// TIA Portal V17 export
// export: Created 2023-02-13T11:16:28.8867509Z, ExportSetting WithDefaults, DisplayName Totally Integrated Automation Portal, DisplayVersion V17, DisplayName TIA Portal Openness, DisplayVersion V17, DisplayName TIA Portal Teamcenter Gateway, DisplayVersion V17, DisplayName TIA Portal Version Control Interface, DisplayVersion V17, DisplayName SINAMICS Startdrive Advanced, DisplayVersion V17, DisplayName SINAMICS Startdrive G130, G150, S120, S150, SINAMICS MV, S210, DisplayVersion V17, DisplayName SINAMICS Startdrive G110M, G120, G120C, G120D, G120P, G115D, DisplayVersion V17, DisplayName STEP 7 Professional, DisplayVersion V17, DisplayName STEP 7 Safety, DisplayVersion V17, DisplayName WinCC Professional, DisplayVersion V17
FUNCTION_BLOCK "IO Digital Preparation"   // FB8, LAD
{ S7_Optimized_Access := 'FALSE' }
VERSION : 0.1
// stored: AutoNumber true, IsIECCheckEnabled false, SetENOAutomatically false, UDAEnableTagReadback false
   VAR_INPUT
      init : Bool;
      Reset : Bool;
   END_VAR
   VAR
      "FS-01.01" { S7_SetPoint := 'True'} : "Digital";   // FLOW SWITCH LINE HOT WATER PHE-01.01
      "DRP-P02.01" { S7_SetPoint := 'True'} : "Digital";   // DRY RUN PROTECTION MONO PUMP P-02.01
      "DRP-P02.02" { S7_SetPoint := 'True'} : "Digital";   // DRY RUN PROTECTION MONO PUMP P-02.03
      "DRP-P03.01" { S7_SetPoint := 'True'} : "Digital";   // DRY RUN PROTECTION MONO PUMP P-03.01
      "DRP-P03.02" { S7_SetPoint := 'True'} : "Digital";   // DRY RUN PROTECTION MONO PUMP P-03.03
      "DRP-P04.01" { S7_SetPoint := 'True'} : "Digital";   // DRY RUN PROTECTION MONO PUMP P-04.01
      "DRP-P05.01" { S7_SetPoint := 'True'} : "Digital";   // DRY RUN PROTECTION MONO PUMP P-05.01
      "DRP-P05.02" { S7_SetPoint := 'True'} : "Digital";   // DRY RUN PROTECTION MONO PUMP P-05.03
      "DRP-P06.01" { S7_SetPoint := 'True'} : "Digital";   // DRY RUN PROTECTION MONO PUMP P-06.01
      "DRP-P07.01" { S7_SetPoint := 'True'} : "Digital";   // DRY RUN PROTECTION MONO PUMP P-07.01
      "DRP-P08.01" { S7_SetPoint := 'True'} : "Digital";   // DRY RUN PROTECTION MONO PUMP P-08.01
      "DRP-P09.01" { S7_SetPoint := 'True'} : "Digital";   // DRY RUN PROTECTION MONO PUMP P-09.01
      "DRP-P09.02" { S7_SetPoint := 'True'} : "Digital";   // DRY RUN PROTECTION MONO PUMP P-09.03
      "LL-51.01" { S7_SetPoint := 'True'} : "Digital";
      "ML-51.01" { S7_SetPoint := 'True'} : "Digital";
      "HL-51.01" { S7_SetPoint := 'True'} : "Digital";
   END_VAR
BEGIN

REGION Network 1: FS-01.01
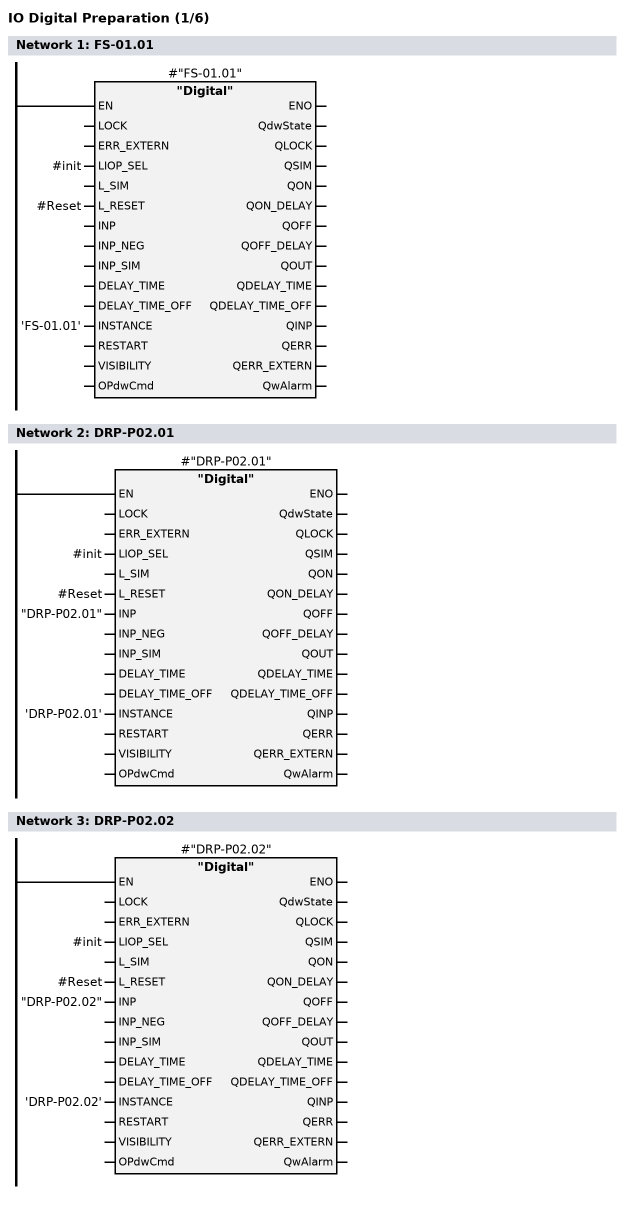
   RUNG wire#powerrail
      #"FS-01.01"(LOCK :=, ERR_EXTERN :=, LIOP_SEL := #init, L_SIM :=, L_RESET := #Reset, INP :=, INP_NEG :=, INP_SIM :=, DELAY_TIME :=, DELAY_TIME_OFF :=, INSTANCE := 'FS-01.01', RESTART :=, VISIBILITY :=, OPdwCmd :=, QdwState =>, QLOCK =>, QSIM =>, QON =>, QON_DELAY =>, QOFF =>, QOFF_DELAY =>, QOUT =>, QDELAY_TIME =>, QDELAY_TIME_OFF =>, QINP =>, QERR =>, QERR_EXTERN =>, QwAlarm =>)
   END_RUNG
   // the same network as SCL:
   #"FS-01.01"(LIOP_SEL := #init, L_RESET := #Reset, INSTANCE := 'FS-01.01');   // "Digital"
END_REGION

REGION Network 2: DRP-P02.01
   RUNG wire#powerrail
      #"DRP-P02.01"(LOCK :=, ERR_EXTERN :=, LIOP_SEL := #init, L_SIM :=, L_RESET := #Reset, INP := "DRP-P02.01", INP_NEG :=, INP_SIM :=, DELAY_TIME :=, DELAY_TIME_OFF :=, INSTANCE := 'DRP-P02.01', RESTART :=, VISIBILITY :=, OPdwCmd :=, QdwState =>, QLOCK =>, QSIM =>, QON =>, QON_DELAY =>, QOFF =>, QOFF_DELAY =>, QOUT =>, QDELAY_TIME =>, QDELAY_TIME_OFF =>, QINP =>, QERR =>, QERR_EXTERN =>, QwAlarm =>)
   END_RUNG
   // the same network as SCL:
   #"DRP-P02.01"(LIOP_SEL := #init, L_RESET := #Reset, INP := "DRP-P02.01", INSTANCE := 'DRP-P02.01');   // "Digital"
END_REGION

REGION Network 3: DRP-P02.02
   RUNG wire#powerrail
      #"DRP-P02.02"(LOCK :=, ERR_EXTERN :=, LIOP_SEL := #init, L_SIM :=, L_RESET := #Reset, INP := "DRP-P02.02", INP_NEG :=, INP_SIM :=, DELAY_TIME :=, DELAY_TIME_OFF :=, INSTANCE := 'DRP-P02.02', RESTART :=, VISIBILITY :=, OPdwCmd :=, QdwState =>, QLOCK =>, QSIM =>, QON =>, QON_DELAY =>, QOFF =>, QOFF_DELAY =>, QOUT =>, QDELAY_TIME =>, QDELAY_TIME_OFF =>, QINP =>, QERR =>, QERR_EXTERN =>, QwAlarm =>)
   END_RUNG
   // the same network as SCL:
   #"DRP-P02.02"(LIOP_SEL := #init, L_RESET := #Reset, INP := "DRP-P02.02", INSTANCE := 'DRP-P02.02');   // "Digital"
END_REGION

REGION Network 4: DRP-P03.01
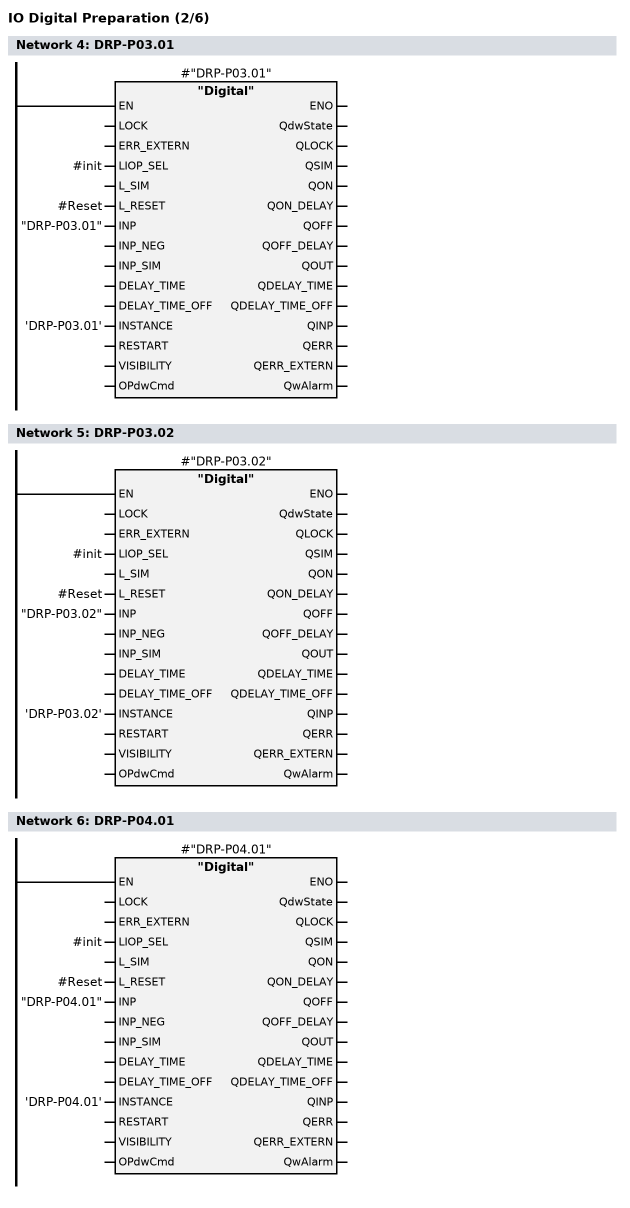
   RUNG wire#powerrail
      #"DRP-P03.01"(LOCK :=, ERR_EXTERN :=, LIOP_SEL := #init, L_SIM :=, L_RESET := #Reset, INP := "DRP-P03.01", INP_NEG :=, INP_SIM :=, DELAY_TIME :=, DELAY_TIME_OFF :=, INSTANCE := 'DRP-P03.01', RESTART :=, VISIBILITY :=, OPdwCmd :=, QdwState =>, QLOCK =>, QSIM =>, QON =>, QON_DELAY =>, QOFF =>, QOFF_DELAY =>, QOUT =>, QDELAY_TIME =>, QDELAY_TIME_OFF =>, QINP =>, QERR =>, QERR_EXTERN =>, QwAlarm =>)
   END_RUNG
   // the same network as SCL:
   #"DRP-P03.01"(LIOP_SEL := #init, L_RESET := #Reset, INP := "DRP-P03.01", INSTANCE := 'DRP-P03.01');   // "Digital"
END_REGION

REGION Network 5: DRP-P03.02
   RUNG wire#powerrail
      #"DRP-P03.02"(LOCK :=, ERR_EXTERN :=, LIOP_SEL := #init, L_SIM :=, L_RESET := #Reset, INP := "DRP-P03.02", INP_NEG :=, INP_SIM :=, DELAY_TIME :=, DELAY_TIME_OFF :=, INSTANCE := 'DRP-P03.02', RESTART :=, VISIBILITY :=, OPdwCmd :=, QdwState =>, QLOCK =>, QSIM =>, QON =>, QON_DELAY =>, QOFF =>, QOFF_DELAY =>, QOUT =>, QDELAY_TIME =>, QDELAY_TIME_OFF =>, QINP =>, QERR =>, QERR_EXTERN =>, QwAlarm =>)
   END_RUNG
   // the same network as SCL:
   #"DRP-P03.02"(LIOP_SEL := #init, L_RESET := #Reset, INP := "DRP-P03.02", INSTANCE := 'DRP-P03.02');   // "Digital"
END_REGION

REGION Network 6: DRP-P04.01
   RUNG wire#powerrail
      #"DRP-P04.01"(LOCK :=, ERR_EXTERN :=, LIOP_SEL := #init, L_SIM :=, L_RESET := #Reset, INP := "DRP-P04.01", INP_NEG :=, INP_SIM :=, DELAY_TIME :=, DELAY_TIME_OFF :=, INSTANCE := 'DRP-P04.01', RESTART :=, VISIBILITY :=, OPdwCmd :=, QdwState =>, QLOCK =>, QSIM =>, QON =>, QON_DELAY =>, QOFF =>, QOFF_DELAY =>, QOUT =>, QDELAY_TIME =>, QDELAY_TIME_OFF =>, QINP =>, QERR =>, QERR_EXTERN =>, QwAlarm =>)
   END_RUNG
   // the same network as SCL:
   #"DRP-P04.01"(LIOP_SEL := #init, L_RESET := #Reset, INP := "DRP-P04.01", INSTANCE := 'DRP-P04.01');   // "Digital"
END_REGION

REGION Network 7: DRP-P05.01
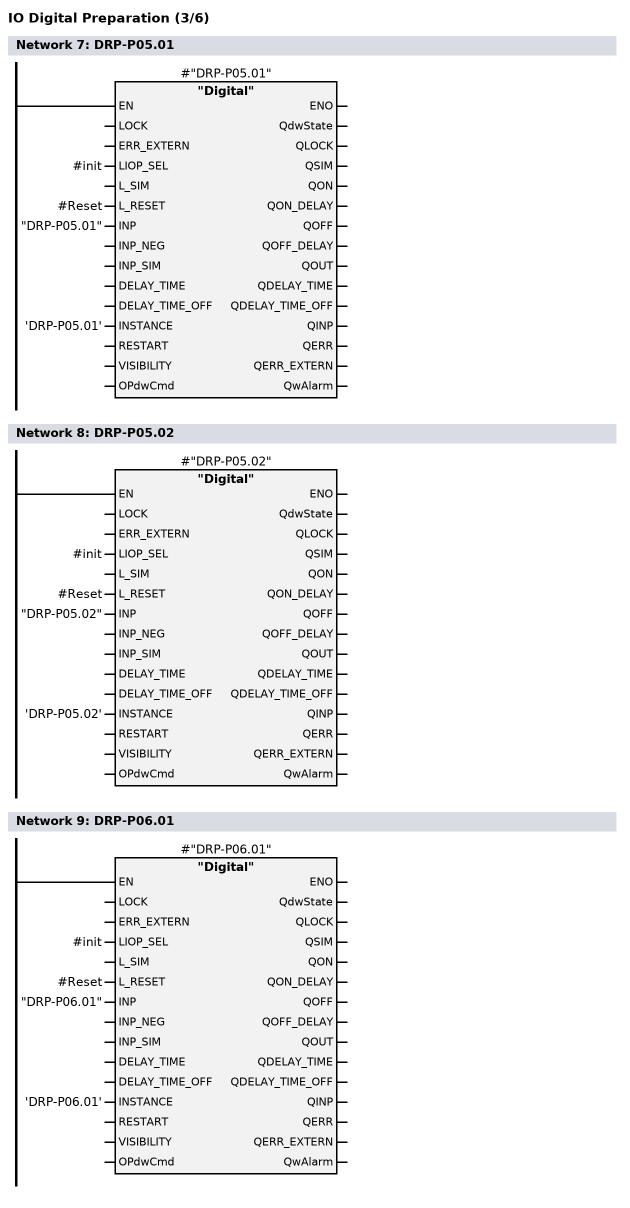
   RUNG wire#powerrail
      #"DRP-P05.01"(LOCK :=, ERR_EXTERN :=, LIOP_SEL := #init, L_SIM :=, L_RESET := #Reset, INP := "DRP-P05.01", INP_NEG :=, INP_SIM :=, DELAY_TIME :=, DELAY_TIME_OFF :=, INSTANCE := 'DRP-P05.01', RESTART :=, VISIBILITY :=, OPdwCmd :=, QdwState =>, QLOCK =>, QSIM =>, QON =>, QON_DELAY =>, QOFF =>, QOFF_DELAY =>, QOUT =>, QDELAY_TIME =>, QDELAY_TIME_OFF =>, QINP =>, QERR =>, QERR_EXTERN =>, QwAlarm =>)
   END_RUNG
   // the same network as SCL:
   #"DRP-P05.01"(LIOP_SEL := #init, L_RESET := #Reset, INP := "DRP-P05.01", INSTANCE := 'DRP-P05.01');   // "Digital"
END_REGION

REGION Network 8: DRP-P05.02
   RUNG wire#powerrail
      #"DRP-P05.02"(LOCK :=, ERR_EXTERN :=, LIOP_SEL := #init, L_SIM :=, L_RESET := #Reset, INP := "DRP-P05.02", INP_NEG :=, INP_SIM :=, DELAY_TIME :=, DELAY_TIME_OFF :=, INSTANCE := 'DRP-P05.02', RESTART :=, VISIBILITY :=, OPdwCmd :=, QdwState =>, QLOCK =>, QSIM =>, QON =>, QON_DELAY =>, QOFF =>, QOFF_DELAY =>, QOUT =>, QDELAY_TIME =>, QDELAY_TIME_OFF =>, QINP =>, QERR =>, QERR_EXTERN =>, QwAlarm =>)
   END_RUNG
   // the same network as SCL:
   #"DRP-P05.02"(LIOP_SEL := #init, L_RESET := #Reset, INP := "DRP-P05.02", INSTANCE := 'DRP-P05.02');   // "Digital"
END_REGION

REGION Network 9: DRP-P06.01
   RUNG wire#powerrail
      #"DRP-P06.01"(LOCK :=, ERR_EXTERN :=, LIOP_SEL := #init, L_SIM :=, L_RESET := #Reset, INP := "DRP-P06.01", INP_NEG :=, INP_SIM :=, DELAY_TIME :=, DELAY_TIME_OFF :=, INSTANCE := 'DRP-P06.01', RESTART :=, VISIBILITY :=, OPdwCmd :=, QdwState =>, QLOCK =>, QSIM =>, QON =>, QON_DELAY =>, QOFF =>, QOFF_DELAY =>, QOUT =>, QDELAY_TIME =>, QDELAY_TIME_OFF =>, QINP =>, QERR =>, QERR_EXTERN =>, QwAlarm =>)
   END_RUNG
   // the same network as SCL:
   #"DRP-P06.01"(LIOP_SEL := #init, L_RESET := #Reset, INP := "DRP-P06.01", INSTANCE := 'DRP-P06.01');   // "Digital"
END_REGION

REGION Network 10: DRP-P07.01
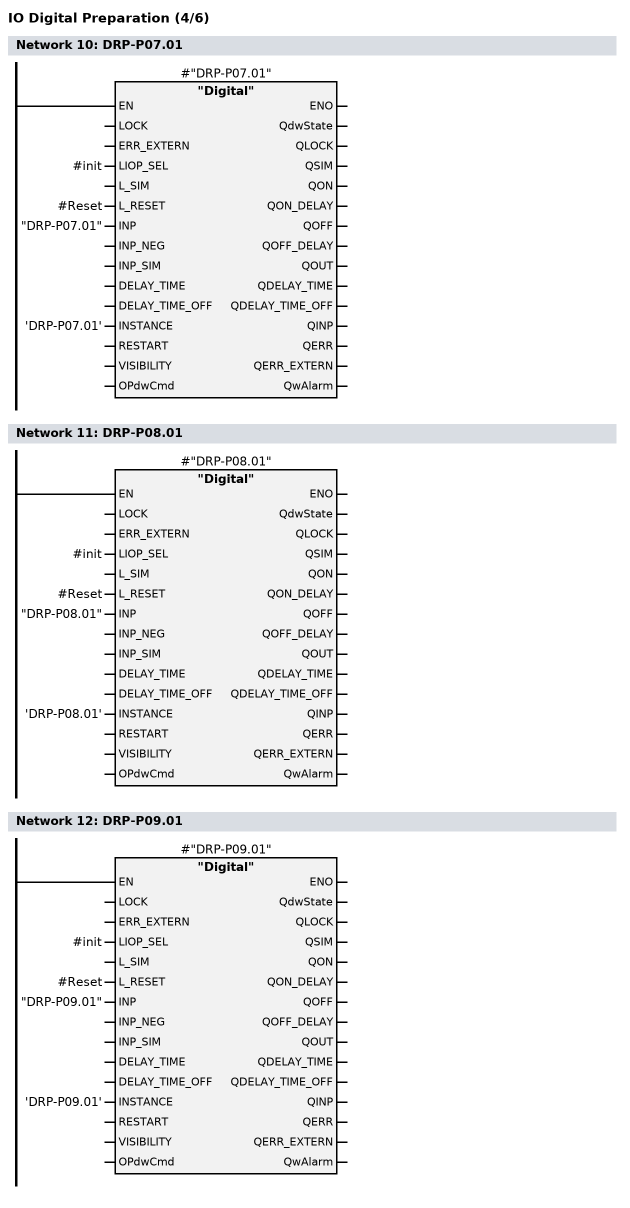
   RUNG wire#powerrail
      #"DRP-P07.01"(LOCK :=, ERR_EXTERN :=, LIOP_SEL := #init, L_SIM :=, L_RESET := #Reset, INP := "DRP-P07.01", INP_NEG :=, INP_SIM :=, DELAY_TIME :=, DELAY_TIME_OFF :=, INSTANCE := 'DRP-P07.01', RESTART :=, VISIBILITY :=, OPdwCmd :=, QdwState =>, QLOCK =>, QSIM =>, QON =>, QON_DELAY =>, QOFF =>, QOFF_DELAY =>, QOUT =>, QDELAY_TIME =>, QDELAY_TIME_OFF =>, QINP =>, QERR =>, QERR_EXTERN =>, QwAlarm =>)
   END_RUNG
   // the same network as SCL:
   #"DRP-P07.01"(LIOP_SEL := #init, L_RESET := #Reset, INP := "DRP-P07.01", INSTANCE := 'DRP-P07.01');   // "Digital"
END_REGION

REGION Network 11: DRP-P08.01
   RUNG wire#powerrail
      #"DRP-P08.01"(LOCK :=, ERR_EXTERN :=, LIOP_SEL := #init, L_SIM :=, L_RESET := #Reset, INP := "DRP-P08.01", INP_NEG :=, INP_SIM :=, DELAY_TIME :=, DELAY_TIME_OFF :=, INSTANCE := 'DRP-P08.01', RESTART :=, VISIBILITY :=, OPdwCmd :=, QdwState =>, QLOCK =>, QSIM =>, QON =>, QON_DELAY =>, QOFF =>, QOFF_DELAY =>, QOUT =>, QDELAY_TIME =>, QDELAY_TIME_OFF =>, QINP =>, QERR =>, QERR_EXTERN =>, QwAlarm =>)
   END_RUNG
   // the same network as SCL:
   #"DRP-P08.01"(LIOP_SEL := #init, L_RESET := #Reset, INP := "DRP-P08.01", INSTANCE := 'DRP-P08.01');   // "Digital"
END_REGION

REGION Network 12: DRP-P09.01
   RUNG wire#powerrail
      #"DRP-P09.01"(LOCK :=, ERR_EXTERN :=, LIOP_SEL := #init, L_SIM :=, L_RESET := #Reset, INP := "DRP-P09.01", INP_NEG :=, INP_SIM :=, DELAY_TIME :=, DELAY_TIME_OFF :=, INSTANCE := 'DRP-P09.01', RESTART :=, VISIBILITY :=, OPdwCmd :=, QdwState =>, QLOCK =>, QSIM =>, QON =>, QON_DELAY =>, QOFF =>, QOFF_DELAY =>, QOUT =>, QDELAY_TIME =>, QDELAY_TIME_OFF =>, QINP =>, QERR =>, QERR_EXTERN =>, QwAlarm =>)
   END_RUNG
   // the same network as SCL:
   #"DRP-P09.01"(LIOP_SEL := #init, L_RESET := #Reset, INP := "DRP-P09.01", INSTANCE := 'DRP-P09.01');   // "Digital"
END_REGION

REGION Network 13: DRP-P09.02
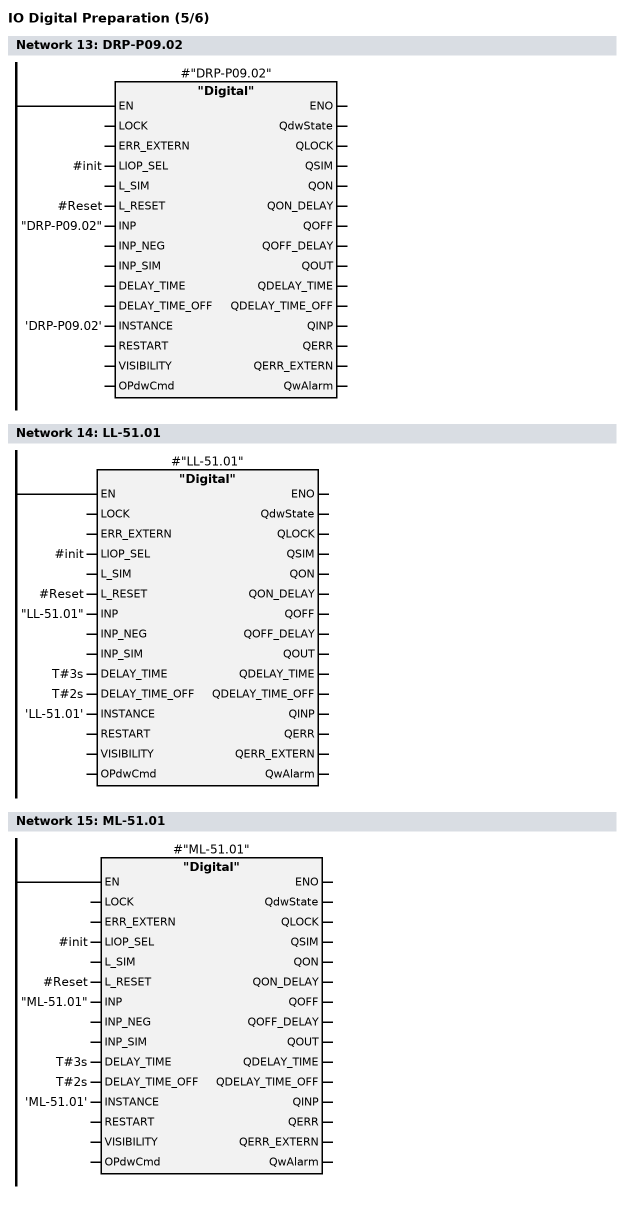
   RUNG wire#powerrail
      #"DRP-P09.02"(LOCK :=, ERR_EXTERN :=, LIOP_SEL := #init, L_SIM :=, L_RESET := #Reset, INP := "DRP-P09.02", INP_NEG :=, INP_SIM :=, DELAY_TIME :=, DELAY_TIME_OFF :=, INSTANCE := 'DRP-P09.02', RESTART :=, VISIBILITY :=, OPdwCmd :=, QdwState =>, QLOCK =>, QSIM =>, QON =>, QON_DELAY =>, QOFF =>, QOFF_DELAY =>, QOUT =>, QDELAY_TIME =>, QDELAY_TIME_OFF =>, QINP =>, QERR =>, QERR_EXTERN =>, QwAlarm =>)
   END_RUNG
   // the same network as SCL:
   #"DRP-P09.02"(LIOP_SEL := #init, L_RESET := #Reset, INP := "DRP-P09.02", INSTANCE := 'DRP-P09.02');   // "Digital"
END_REGION

REGION Network 14: LL-51.01
   RUNG wire#powerrail
      #"LL-51.01"(LOCK :=, ERR_EXTERN :=, LIOP_SEL := #init, L_SIM :=, L_RESET := #Reset, INP := "LL-51.01", INP_NEG :=, INP_SIM :=, DELAY_TIME := T#3s, DELAY_TIME_OFF := T#2s, INSTANCE := 'LL-51.01', RESTART :=, VISIBILITY :=, OPdwCmd :=, QdwState =>, QLOCK =>, QSIM =>, QON =>, QON_DELAY =>, QOFF =>, QOFF_DELAY =>, QOUT =>, QDELAY_TIME =>, QDELAY_TIME_OFF =>, QINP =>, QERR =>, QERR_EXTERN =>, QwAlarm =>)
   END_RUNG
   // the same network as SCL:
   #"LL-51.01"(LIOP_SEL := #init,   // "Digital"
               L_RESET := #Reset,
               INP := "LL-51.01",
               DELAY_TIME := T#3s,
               DELAY_TIME_OFF := T#2s,
               INSTANCE := 'LL-51.01');
END_REGION

REGION Network 15: ML-51.01
   RUNG wire#powerrail
      #"ML-51.01"(LOCK :=, ERR_EXTERN :=, LIOP_SEL := #init, L_SIM :=, L_RESET := #Reset, INP := "ML-51.01", INP_NEG :=, INP_SIM :=, DELAY_TIME := T#3s, DELAY_TIME_OFF := T#2s, INSTANCE := 'ML-51.01', RESTART :=, VISIBILITY :=, OPdwCmd :=, QdwState =>, QLOCK =>, QSIM =>, QON =>, QON_DELAY =>, QOFF =>, QOFF_DELAY =>, QOUT =>, QDELAY_TIME =>, QDELAY_TIME_OFF =>, QINP =>, QERR =>, QERR_EXTERN =>, QwAlarm =>)
   END_RUNG
   // the same network as SCL:
   #"ML-51.01"(LIOP_SEL := #init,   // "Digital"
               L_RESET := #Reset,
               INP := "ML-51.01",
               DELAY_TIME := T#3s,
               DELAY_TIME_OFF := T#2s,
               INSTANCE := 'ML-51.01');
END_REGION

REGION Network 16: HL-51.01
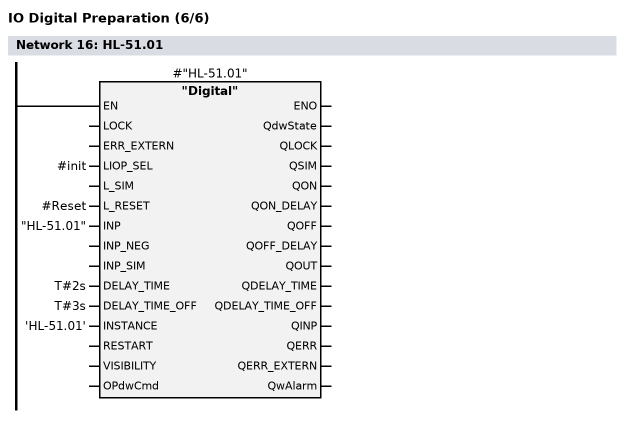
   RUNG wire#powerrail
      #"HL-51.01"(LOCK :=, ERR_EXTERN :=, LIOP_SEL := #init, L_SIM :=, L_RESET := #Reset, INP := "HL-51.01", INP_NEG :=, INP_SIM :=, DELAY_TIME := T#2s, DELAY_TIME_OFF := T#3s, INSTANCE := 'HL-51.01', RESTART :=, VISIBILITY :=, OPdwCmd :=, QdwState =>, QLOCK =>, QSIM =>, QON =>, QON_DELAY =>, QOFF =>, QOFF_DELAY =>, QOUT =>, QDELAY_TIME =>, QDELAY_TIME_OFF =>, QINP =>, QERR =>, QERR_EXTERN =>, QwAlarm =>)
   END_RUNG
   // the same network as SCL:
   #"HL-51.01"(LIOP_SEL := #init,   // "Digital"
               L_RESET := #Reset,
               INP := "HL-51.01",
               DELAY_TIME := T#2s,
               DELAY_TIME_OFF := T#3s,
               INSTANCE := 'HL-51.01');
END_REGION
END_FUNCTION_BLOCK
